Fanuc KAREL source: kd00001.KL

-- PROVISIONAL review KL for V1013-1; original PC SHA256 d611a98c8c1dfdb16d5efd6796a0eaad80d11e35137c25fa5c71cd51c00cc8e3
-- Incomplete behavior may be omitted. Consult companion uncertainty JSON. Do not deploy.
PROGRAM KD00001
%NOLOCKGROUP
VAR
  I : INTEGER
  J : INTEGER
  B : BOOLEAN
  R : REAL
  S : STRING[80]
BEGIN
  -- UNRESOLVED_PC offsets 5-12; opcodes 9D,23
  -- UNRESOLVED_PC offsets 17-21; opcodes 7F
END KD00001
